PROGRAM _18_Otros_Operadores2


QUERYPOINTER();
TRY_CATCH();
VARINFO();
TestAndSet1();

END_PROGRAM

(* stored: Version 1.1.0.1, ProductVersion 3.1.4024.12
   POU _18_Otros_Operadores2: Id {00ab3834-d803-4525-b9eb-d217f66d4b14}, SpecialFunc None *)
